PROGRAM MAIN
VAR
END_VAR

END_PROGRAM

(* stored: Version 1.1.0.1
   POU MAIN: Id {ae9a17d4-c04a-4a4f-a5a1-07c9c1e54e8b} *)
